PROGRAM POU
VAR
	btest: BOOL;
END_VAR

btest := TRUE;

END_PROGRAM

(* stored: Version 1.1.0.1, ProductVersion 3.1.4024.15
   POU POU: Id {3fc62ccb-fe41-4ede-9fd5-674cbea254bf}, SpecialFunc None *)
